// TIA Portal V16 export
// export: Created 2021-04-06T19:52:19.9784212Z, ExportSetting WithDefaults, DisplayName Totally Integrated Automation Portal, DisplayVersion V16, DisplayName TIA Portal Version Control Interface, DisplayVersion V16, DisplayName TIA Portal Openness, DisplayVersion V16, DisplayName STEP 7 Professional, DisplayVersion V16, DisplayName STEP 7 Safety, DisplayVersion V16, DisplayName WinCC Unified SCADA Engineering System, DisplayVersion V16
TYPE "mode"
// stored: IsFailsafeCompliant false
   STRUCT
      Yq_ReadyDoze : Array[0..2] of Bool;
      Conv_FRV : Array[0..2] of Bool;   // Конвейер1 - вперед
      Conv_REV : Array[0..2] of Bool;   // Конвейер1 - назад
      Door_open : Array[0..12] of Bool;   // Лопатка - открыть
      Door_close : Array[0..12] of Bool;   // Лопатка - закрыть
      Bunker_leftOpen : Array[0..12] of Bool;   // Бункер - открыть влево
      Bunker_leftClose : Array[0..12] of Bool;   // Бункер - закрыть влево
      Bunker_rightOpen : Array[0..12] of Bool;   // Бункер - открыть вправо
      Bunker_rightClose : Array[0..12] of Bool;   // Бункер - закрыть вправо
      flipper_Up : Bool;   // управление плавником вверх
      flipper_Down : Bool;   // управление плавником вниз
      vibroTable : Array[0..2] of Bool;   // управление вибростолом
      vibroLot : Array[0..12] of Bool;   // управление вибролотком
      setVibration : Real;   // уставка вибрации
      setSpeedInConv : Real;   // скорость питателя
      startInConv : Bool;   // запуск питателя
   END_STRUCT;
END_TYPE
